% RSLogix 500 project I2P-JOB-13B-MITCH_BAK056.RSS, saved by version 10.00.00.00 %
PROJECT "ML01B"    % processor: Bul.1763 MicroLogix 1100 Series B %

PROGRAM FILES
  LAD 2   13 rungs

DATA FILES
  O0 OUTPUT  4 elements
  I1 INPUT  6 elements
  S2 STATUS  66 elements
  B3 BINARY  1 elements
  T4 TIMER  1 elements
  C5 COUNTER  1 elements
  R6 CONTROL  1 elements
  N7 INTEGER  1 elements
  F8 FLOAT  1 elements

LADDER 2
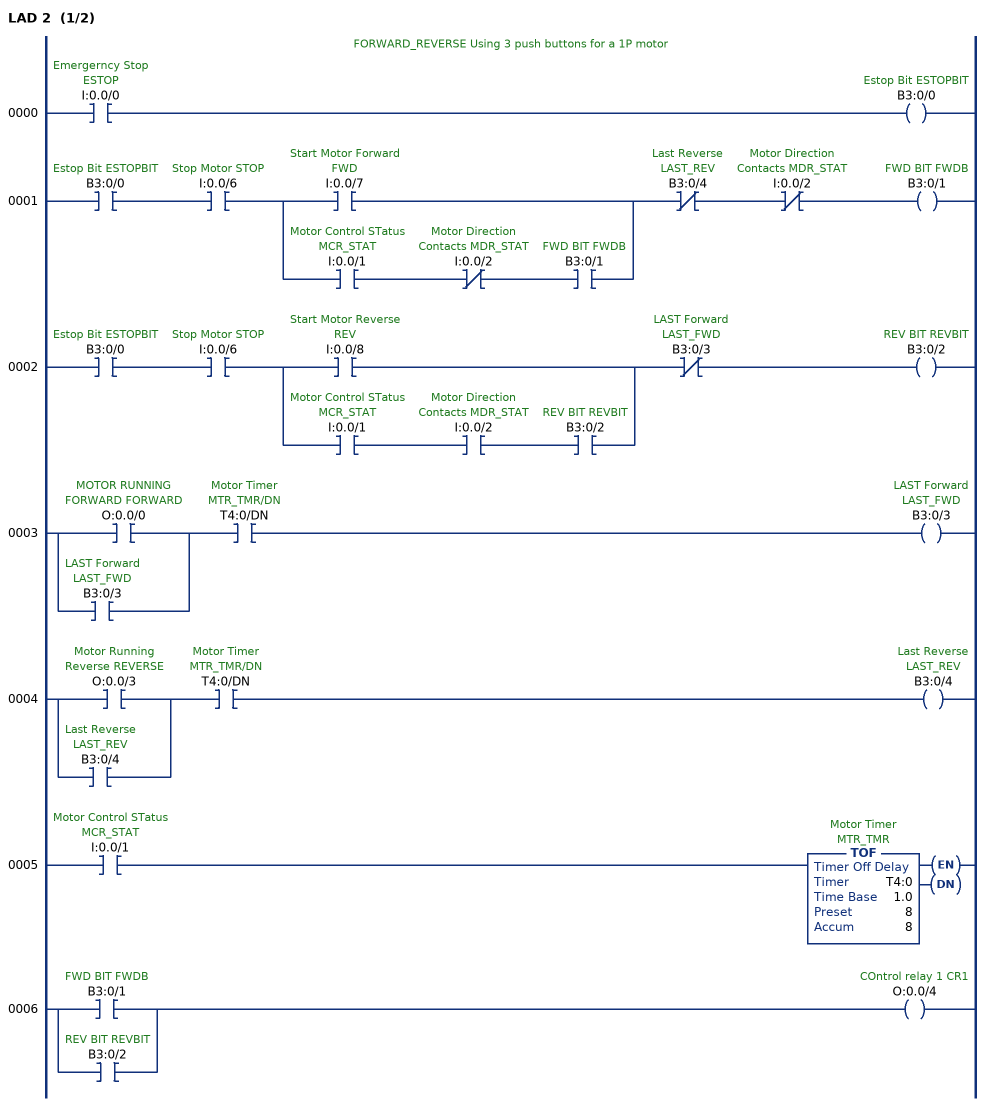
% Rung: 0 %
% FORWARD_REVERSE Using 3 push buttons for a 1P motor %
SOR XIC I:0.0/0 OTE B3:0/0 EOR
%   I:0.0/0  ESTOP  "Emergerncy Stop" %
%   B3:0/0  ESTOPBIT  "Estop Bit" %
% Rung: 1 %
SOR XIC B3:0/0 XIC I:0.0/6 BST XIC I:0.0/7 NXB XIC I:0.0/1 XIO I:0.0/2 XIC B3:0/1 BND XIO B3:0/4 XIO I:0.0/2 OTE B3:0/1 EOR
%   B3:0/0  ESTOPBIT  "Estop Bit" %
%   I:0.0/6  STOP  "Stop Motor" %
%   I:0.0/7  FWD  "Start Motor Forward" %
%   I:0.0/1  MCR_STAT  "Motor Control STatus" %
%   I:0.0/2  MDR_STAT  "Motor Direction Contacts" %
%   B3:0/1  FWDB  "FWD BIT" %
%   B3:0/4  LAST_REV  "Last Reverse" %
% Rung: 2 %
SOR XIC B3:0/0 XIC I:0.0/6 BST XIC I:0.0/8 NXB XIC I:0.0/1 XIC I:0.0/2 XIC B3:0/2 BND XIO B3:0/3 OTE B3:0/2 EOR
%   B3:0/0  ESTOPBIT  "Estop Bit" %
%   I:0.0/6  STOP  "Stop Motor" %
%   I:0.0/8  REV  "Start Motor Reverse" %
%   I:0.0/1  MCR_STAT  "Motor Control STatus" %
%   I:0.0/2  MDR_STAT  "Motor Direction Contacts" %
%   B3:0/2  REVBIT  "REV BIT" %
%   B3:0/3  LAST_FWD  "LAST Forward" %
% Rung: 3 %
SOR BST XIC O:0.0/0 NXB XIC B3:0/3 BND XIC T4:0/DN OTE B3:0/3 EOR
%   O:0.0/0  FORWARD  "MOTOR RUNNING FORWARD" %
%   B3:0/3  LAST_FWD  "LAST Forward" %
%   T4:0  MTR_TMR  "Motor Timer" %
% Rung: 4 %
SOR BST XIC O:0.0/3 NXB XIC B3:0/4 BND XIC T4:0/DN OTE B3:0/4 EOR
%   O:0.0/3  REVERSE  "Motor Running Reverse" %
%   B3:0/4  LAST_REV  "Last Reverse" %
%   T4:0  MTR_TMR  "Motor Timer" %
% Rung: 5 %
SOR XIC I:0.0/1 TOF T4:0 1.0 8 8 EOR
%   I:0.0/1  MCR_STAT  "Motor Control STatus" %
%   T4:0  MTR_TMR  "Motor Timer" %
% Rung: 6 %
SOR BST XIC B3:0/1 NXB XIC B3:0/2 BND OTE O:0.0/4 EOR
%   B3:0/1  FWDB  "FWD BIT" %
%   B3:0/2  REVBIT  "REV BIT" %
%   O:0.0/4  CR1  "COntrol relay 1" %

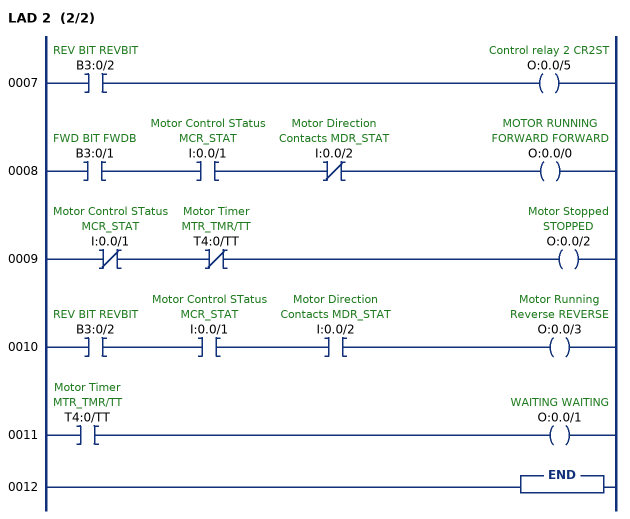
% Rung: 7 %
SOR XIC B3:0/2 OTE O:0.0/5 EOR
%   B3:0/2  REVBIT  "REV BIT" %
%   O:0.0/5  CR2ST  "Control relay 2" %
% Rung: 8 %
SOR XIC B3:0/1 XIC I:0.0/1 XIO I:0.0/2 OTE O:0.0/0 EOR
%   B3:0/1  FWDB  "FWD BIT" %
%   I:0.0/1  MCR_STAT  "Motor Control STatus" %
%   I:0.0/2  MDR_STAT  "Motor Direction Contacts" %
%   O:0.0/0  FORWARD  "MOTOR RUNNING FORWARD" %
% Rung: 9 %
SOR XIO I:0.0/1 XIO T4:0/TT OTE O:0.0/2 EOR
%   I:0.0/1  MCR_STAT  "Motor Control STatus" %
%   T4:0  MTR_TMR  "Motor Timer" %
%   O:0.0/2  STOPPED  "Motor Stopped" %
% Rung: 10 %
SOR XIC B3:0/2 XIC I:0.0/1 XIC I:0.0/2 OTE O:0.0/3 EOR
%   B3:0/2  REVBIT  "REV BIT" %
%   I:0.0/1  MCR_STAT  "Motor Control STatus" %
%   I:0.0/2  MDR_STAT  "Motor Direction Contacts" %
%   O:0.0/3  REVERSE  "Motor Running Reverse" %
% Rung: 11 %
SOR XIC T4:0/TT OTE O:0.0/1 EOR
%   T4:0  MTR_TMR  "Motor Timer" %
%   O:0.0/1  WAITING  "WAITING" %
% Rung: 12 %
SOR END EOR

OTHER DOCUMENTED ADDRESSES
  I:0.0/3  DIRECTION  "Direction Forward- off-Reverse"
  I:0.0/4  3PSS_B  "Three posision selector switch B"
  I:0.0/5  2PSSA  "2 position selector switch A"
  T4:1/TT  TT

DATA TABLE (non-zero values as saved)
DATA B3
% B3:0 % 0X0001
DATA T4
% .PRE .ACC %
% T4:0 % 8 8
